{attribute 'linkalways'} 
{attribute 'no_explicit_call' := 'This FB is a CLASS and must be accessed using methods or properties'}
{attribute 'enable_dynamic_creation'}
FUNCTION_BLOCK Node_F_VN_SetRoi_TcVnRectangle_UDINT EXTENDS VisionNode
VAR
    stRoi : _TcVnRectangle_UDINT;
    ipDestImage : _ITcVnImage;
    hrPrev : _HRESULT(S_OK);
	hresult : _HRESULT(S_OK);
END_VAR

METHOD PUBLIC  Clone : I_Node
VAR
	pNode : POINTER TO Node_F_VN_SetRoi_TcVnRectangle_UDINT;
END_VAR
pNode := __NEW(Node_F_VN_SetRoi_TcVnRectangle_UDINT);
Clone := pNode^;
END_METHOD

METHOD FB_init : BOOL
VAR_INPUT
	bInitRetains : BOOL; // if TRUE, the retain variables are initialized (warm start / cold start)
	bInCopyCode : BOOL;  // if TRUE, the instance afterwards gets moved into the copy code (online change)
END_VAR
AddInput('stRoi', stRoi);
AddInput('ipDestImage', ipDestImage);
AddInput('hrPrev', hrPrev);
AddOutput('ipDestImage', ipDestImage);
AddOutput('hresult',hresult);
END_METHOD

METHOD PROTECTED OnExecute
hresult.Value := F_VN_SetRoi_TcVnRectangle_UDINT(
    stRoi := stRoi.Value,
	ipDestImage := ipDestImage.Value,
	hrPrev:= hrPrev.Value);
END_METHOD

METHOD PUBLIC PreExecutionCheck
VAR_INPUT
	Check : I_PreExecutionChecks;
END_VAR
VAR
    imageWidth : UDINT;
    imageHeight : UDINT;
END_VAR
Check.IsTrue(ipDestImage.IsValid, 'ipDestImage must contain an image');

IF Check.Failed THEN
    RETURN;
END_IF

ipDestImage.Value.GetWidth(imageWidth);
ipDestImage.Value.GetHeight(imageHeight);

Check.IsTrue(IsRoiSizeOK_Udint(stRoi.Value, imageWidth, imageHeight), 'ROI must fit within image');
END_METHOD

END_FUNCTION_BLOCK

(* stored: Version 1.1.0.1, ProductVersion 3.1.4024.13
   POU Node_F_VN_SetRoi_TcVnRectangle_UDINT: Id {3ed9d8d8-40b7-0167-2e31-093cc99a83b8}, SpecialFunc None
   Folder Constructor: Id {b9a314bb-b088-0476-2aec-9fb445d7e274}
   Method Clone: Id {cacf75dd-f619-06b5-091e-91ba36572fed}
   Method FB_init: Id {a6b86ffa-cd3c-065b-2b90-f3c6a263e284}
   Method OnExecute: Id {d9dfee31-3767-0576-1c8c-1afdbc449744}
   Method PreExecutionCheck: Id {3e96d810-bc18-0564-32ab-361c14fc3281} *)
